FUNCTION_BLOCK FB_Slider
VAR_INPUT
END_VAR
VAR_OUTPUT
END_VAR
VAR
END_VAR

END_FUNCTION_BLOCK

(* stored: Version 1.1.0.1, ProductVersion 3.1.4024.14
   POU FB_Slider: Id {981876b1-819e-49a2-9856-6ba956b93924}, SpecialFunc None *)
